FUNCTION_BLOCK JsonTypeConverters IMPLEMENTS I_JsonTypeConverters
VAR
	converters : Dictionary;
END_VAR

METHOD PUBLIC GetByDataType : I_JsonTypeConverter
VAR_INPUT
	DataType : T_MAXSTRING;
END_VAR
converters.TryGetValue(DataType, GetByDataType);
END_METHOD

METHOD PUBLIC HasDataType : BOOL
VAR_INPUT
	DataType : T_MAXSTRING;
END_VAR
HasDataType := converters.ContainsKey(DataType);
END_METHOD

METHOD PUBLIC InsertByDataType
VAR_INPUT
	DataType : T_MAXSTRING;
	TypeConverter : I_JsonTypeConverter;
END_VAR
converters.AddOrUpdate(DataType,TypeConverter);
END_METHOD

END_FUNCTION_BLOCK

(* stored: Version 1.1.0.1, ProductVersion 3.1.4024.12
   POU JsonTypeConverters: Id {695b6b4a-c949-0743-1d47-4a41f3736c15}, SpecialFunc None
   Method GetByDataType: Id {0e472e8b-43d1-041b-35b0-54c91730f712}
   Method HasDataType: Id {e32e9a4b-b30f-0b9b-0b57-3cce473d9857}
   Method InsertByDataType: Id {66c90401-a850-06d1-0c36-79dbafbbe7b4} *)
